Fanuc KAREL source: f_move3_t.kl

PROGRAM F_MOVE3_T
VAR
path1   :PATH
p : POSITION
i : INTEGER
BEGIN
    MOVE TO p,
        WHEN ERROR[*] DO CANCEL
        WHEN DIN[1] AND DIN[2] DO STOP
        WHEN DIN[3] OR ERROR[12] DO PAUSE
    ENDMOVE
    MOVE ALONG path1,
        WHEN AT NODE[2] DO DOUT[1] = TRUE
    ENDMOVE
END F_MOVE3_T
